Yaskawa INFORM job: test2.jbi

/JOB
//NAME TEST2
//POS
///NPOS 0,0,0,0,0,0
//INST
///DATE 2021/01/13 18:20
///ATTR SC,RW
///GROUP1 RB1,ST1
///LVARS 3,3,3,3,0,0,0,0
NOP
IFTHEN IN#(12)=ON
ELSEIF IN#(23)=OFF
   DOUT OG#(12) B012


ENDIF


SET D112 LD123
SET LD123  EXPRESS expression}


SET LD012  EXPRESS LD012 + expression




CNVRT PX001 PX003 RF
CNVRT PX012 PX034 UF#(1) TL#(0)

MFRAME UF#(12) LPX001 LPX002 LPX003


SET LB002 LB123


SET B### B###

SET LD123  EXPRESS ( LI000 + LI001 ) * 1000
SET D123  EXPRESS D000 + ( LI000 + LI001 ) * 1000

SET D123  EXPRESS $2{expression}

SET LD123  EXPRESS ${2:expression}



ELSEIF condition ANDEXP condition}

END
